# EPICS IOC start-up script: crs-c3s_ctrl-plc-01-loc/iocsh/crs-c3s_ctrl-plc-01-test.iocsh
# @field crs-c3s_ctrl-plc-01_VERSION
# @runtime YES

# Load plc interface database
dbLoadRecords("crs-c3s_ctrl-plc-01-test.db", "MODVERSION=$(crs-c3s_ctrl-plc-01_VERSION)")
